// TwinCAT 3 PLC project las_bts
// Title: lcls-plc-las-bts
// Company: SLAC
// ProjectVersion: 1.0.0
// ProgramVersion: 3.1.4023.0
// libraries:
//   LCLSVacuumSerialDriverLib, * (SLAC)
//   Tc2_SerialCom, * (Beckhoff Automation GmbH)
//   Tc2_Standard, * (Beckhoff Automation GmbH)
//   Tc2_System, * (Beckhoff Automation GmbH)
//   Tc2_Utilities, * (Beckhoff Automation GmbH)
//   Tc3_Module, * (Beckhoff Automation GmbH)
//   TcUnit, * (www.tcunit.org)
//   LCLS General,2.4.2,SLAC
//   LCLS Vacuum,2.0.1,SLAC - LCLS
//   PMPS,2.2.1,SLAC - LCLS
// project tree:
//   / ComTask.TcTTO (not stored), PlcTask.TcTTO (not stored)
//   DUTs/ ST_ShutterControl.TcDUT (not stored), ST_SourceDataStore.TcDUT (not stored), ST_EpicsMotorMSTA.TcDUT (not stored)
//   GVLs/ GVL_BTPS.TcGVL (not stored), GVL_BTPS_Constants.TcGVL (not stored), GVL_BTPS_Retain.TcGVL (not stored), GVL_BTS_VAC.TcGVL, GVL_COM.TcGVL (not stored), GVL_Constants.TcGVL (not stored), GVL_Shutters.TcGVL (not stored), GVL_Variables.TcGVL (not stored)
//   POUs/BTPS/ FB_DestinationDataStore.TcPOU (not stored), FB_EpicsMotorMonitor.TcPOU (not stored), FB_EpicsStatsMonitor.TcPOU (not stored), FB_RangeComparison.TcPOU (not stored), FB_ShutterSafety.TcPOU (not stored), F_IsValveReady.TcPOU (not stored)
//   POUs/BTPS/Tests/ FB_TestRangeComparison.TcPOU (not stored), FB_TestShutterSafety.TcPOU (not stored), FB_Test_EpicsCentroidMonitor.TcPOU (not stored), FB_Test_EpicsMotorMonitor.TcPOU (not stored), PRG_RunTests.TcPOU (not stored)
//   POUs/ DIAGNOSTICS.TcPOU (not stored), MAIN.TcPOU (not stored), PRG_BTPS.TcPOU (not stored), PRG_COM.TcPOU (not stored), PRG_GAUGES.TcPOU (not stored), PRG_PUMPS.TcPOU (not stored), PRG_SavePeristentVariables.TcPOU (not stored), PRG_ShutterRequest.TcPOU (not stored), PRG_VALVES.TcPOU
// real-time tasks:
//   TASK PlcTask: cycle T#10ms, priority 20, ADS port 350
//   TASK ComTask: cycle T#11ms, priority 1, ADS port 351
// I/O:
//   DEVICE EtherCAT1
// variable links:
//   las_bts/las_bts Instance <-> EtherCAT1/EK1100_01_00/EL1004_01_16
//     PlcTask Inputs/GVL_BTS_VAC.fb_LS3_PIP.i_xSP_DI <-> Channel 1/Input
//     PlcTask Inputs/GVL_BTS_VAC.fb_LS4_PIP.i_xSP_DI <-> Channel 2/Input
//     PlcTask Inputs/GVL_BTS_VAC.fb_LS6_PIP.i_xSP_DI <-> Channel 3/Input
//   las_bts/las_bts Instance <-> EtherCAT1/EK1100_01_00/EL1124_01_06
//     PlcTask Inputs/GVL_BTS_VAC.fb_LS3_GCC.i_xDisc_Active <-> Channel 4/Input
//     PlcTask Inputs/GVL_BTS_VAC.fb_LS3_GCC.i_xHV_ON <-> Channel 3/Input
//     PlcTask Inputs/GVL_BTS_VAC.fb_PP_GCC.i_xDisc_Active <-> Channel 2/Input
//     PlcTask Inputs/GVL_BTS_VAC.fb_PP_GCC.i_xHV_ON <-> Channel 1/Input
//   las_bts/las_bts Instance <-> EtherCAT1/EK1100_01_00/EL1124_01_07
//     PlcTask Inputs/GVL_BTS_VAC.fb_DP_GCC.i_xDisc_Active <-> Channel 4/Input
//     PlcTask Inputs/GVL_BTS_VAC.fb_DP_GCC.i_xHV_ON <-> Channel 3/Input
//     PlcTask Inputs/GVL_BTS_VAC.fb_LD2_GCC.i_xDisc_Active <-> Channel 2/Input
//     PlcTask Inputs/GVL_BTS_VAC.fb_LD2_GCC.i_xHV_ON <-> Channel 1/Input
//   las_bts/las_bts Instance <-> EtherCAT1/EK1100_01_00/EL1124_01_08
//     PlcTask Inputs/GVL_BTS_VAC.fb_LD8_GCC.i_xDisc_Active <-> Channel 2/Input
//     PlcTask Inputs/GVL_BTS_VAC.fb_LD8_GCC.i_xHV_ON <-> Channel 1/Input
//     PlcTask Inputs/GVL_BTS_VAC.fb_LS4_GCC.i_xDisc_Active <-> Channel 4/Input
//     PlcTask Inputs/GVL_BTS_VAC.fb_LS4_GCC.i_xHV_ON <-> Channel 3/Input
//   las_bts/las_bts Instance <-> EtherCAT1/EK1100_01_00/EL2624_01_01
//     PlcTask Outputs/GVL_BTS_VAC.fb_LD8_GCC.q_xHV_DIS <-> Channel 1/Output
//     PlcTask Outputs/GVL_BTS_VAC.fb_LS3_GCC.q_xHV_DIS <-> Channel 3/Output
//     PlcTask Outputs/GVL_BTS_VAC.fb_LS4_GCC.q_xHV_DIS <-> Channel 4/Output
//   las_bts/las_bts Instance <-> EtherCAT1/EK1100_01_00/EL2624_01_02
//     PlcTask Outputs/GVL_BTS_VAC.fb_DP_GCC.q_xHV_DIS <-> Channel 4/Output
//     PlcTask Outputs/GVL_BTS_VAC.fb_LD2_GCC.q_xHV_DIS <-> Channel 1/Output
//     PlcTask Outputs/GVL_BTS_VAC.fb_PP_GCC.q_xHV_DIS <-> Channel 2/Output
//   las_bts/las_bts Instance <-> EtherCAT1/EK1100_01_00/EL2794_01_17
//     PlcTask Outputs/GVL_BTS_VAC.fb_LS3_PIP.q_xHVEna_DO <-> Channel 1/Output
//     PlcTask Outputs/GVL_BTS_VAC.fb_LS4_PIP.q_xHVEna_DO <-> Channel 2/Output
//     PlcTask Outputs/GVL_BTS_VAC.fb_LS6_PIP.q_xHVEna_DO <-> Channel 3/Output
//   las_bts/las_bts Instance <-> EtherCAT1/EK1100_01_00/EL3064_01_15
//     PlcTask Inputs/GVL_BTS_VAC.fb_LS3_PIP.i_iPRESS <-> AI Standard Channel 1/Value
//     PlcTask Inputs/GVL_BTS_VAC.fb_LS4_PIP.i_iPRESS <-> AI Standard Channel 2/Value
//     PlcTask Inputs/GVL_BTS_VAC.fb_LS6_PIP.i_iPRESS <-> AI Standard Channel 3/Value
//   las_bts/las_bts Instance <-> EtherCAT1/EK1100_01_00/EL3174_01_09
//     PlcTask Inputs/GVL_BTS_VAC.fb_DP_GCC.i_iPRESS_R <-> AI Standard Channel 4/Value
//     PlcTask Inputs/GVL_BTS_VAC.fb_LD2_GCC.i_iPRESS_R <-> AI Standard Channel 1/Value
//     PlcTask Inputs/GVL_BTS_VAC.fb_LS4_GPI.i_iPRESS_R <-> AI Standard Channel 3/Value
//     PlcTask Inputs/GVL_BTS_VAC.fb_LS6_GPI.i_iPRESS_R <-> AI Standard Channel 3/Value
//     PlcTask Inputs/GVL_BTS_VAC.fb_PP_GCC.i_iPRESS_R <-> AI Standard Channel 2/Value
//   las_bts/las_bts Instance <-> EtherCAT1/EK1100_01_00/EL3174_01_10
//     PlcTask Inputs/GVL_BTS_VAC.fb_DP_GPI.i_iPRESS_R <-> AI Standard Channel 2/Value
//     PlcTask Inputs/GVL_BTS_VAC.fb_LD2_GPI.i_iPRESS_R <-> AI Standard Channel 1/Value
//     PlcTask Inputs/GVL_BTS_VAC.fb_LS1_GPI.i_iPRESS_R <-> AI Standard Channel 4/Value
//     PlcTask Inputs/GVL_BTS_VAC.fb_PP_GPI_1.i_iPRESS_R <-> AI Standard Channel 3/Value
//   las_bts/las_bts Instance <-> EtherCAT1/EK1100_01_00/EL3174_01_11
//     PlcTask Inputs/GVL_BTS_VAC.fb_LD8_GCC.i_iPRESS_R <-> AI Standard Channel 3/Value
//     PlcTask Inputs/GVL_BTS_VAC.fb_LD8_GPI.i_iPRESS_R <-> AI Standard Channel 2/Value
//     PlcTask Inputs/GVL_BTS_VAC.fb_LS3_GPI.i_iPRESS_R <-> AI Standard Channel 4/Value
//     PlcTask Inputs/GVL_BTS_VAC.fb_PP_GPI_2.i_iPRESS_R <-> AI Standard Channel 1/Value
//   las_bts/las_bts Instance <-> EtherCAT1/EK1100_01_00/EL3174_01_8A
//     PlcTask Inputs/GVL_BTS_VAC.fb_LS3_GCC.i_iPRESS_R <-> AI Standard Channel 2/Value
//     PlcTask Inputs/GVL_BTS_VAC.fb_LS4_GCC.i_iPRESS_R <-> AI Standard Channel 3/Value
//   las_bts/las_bts Instance <-> EtherCAT1/EK1100_02_00/EL1002_02_01
//     PlcTask Inputs/GVL_BTS_VAC.fb_PP_VRC_1.i_xClsLS <-> Channel 1/Input
//     PlcTask Inputs/GVL_BTS_VAC.fb_PP_VRC_1.i_xOpnLS <-> Channel 2/Input
//   las_bts/las_bts Instance <-> EtherCAT1/EK1100_02_00/EL1002_02_03
//     PlcTask Inputs/GVL_BTS_VAC.fb_PP_VRC_3.i_xClsLS <-> Channel 1/Input
//     PlcTask Inputs/GVL_BTS_VAC.fb_PP_VRC_3.i_xOpnLS <-> Channel 2/Input
//   las_bts/las_bts Instance <-> EtherCAT1/EK1100_02_00/EL1004_02_06
//     PlcTask Inputs/GVL_BTS_VAC.fb_LD9_VGC.i_xClsLS <-> Channel 3/Input
//     PlcTask Inputs/GVL_BTS_VAC.fb_LD9_VGC.i_xOpnLS <-> Channel 4/Input
//     PlcTask Inputs/GVL_BTS_VAC.fb_LS1_VGC.i_xClsLS <-> Channel 1/Input
//     PlcTask Inputs/GVL_BTS_VAC.fb_LS1_VGC.i_xOpnLS <-> Channel 2/Input
//   las_bts/las_bts Instance <-> EtherCAT1/EK1100_02_00/EL1004_02_07
//     PlcTask Inputs/GVL_BTS_VAC.fb_LD10_VGC.i_xClsLS <-> Channel 1/Input
//     PlcTask Inputs/GVL_BTS_VAC.fb_LD8_VGC.i_xClsLS <-> Channel 3/Input
//     PlcTask Inputs/GVL_BTS_VAC.fb_LD10_VGC.i_xOpnLS <-> Channel 2/Input
//     PlcTask Inputs/GVL_BTS_VAC.fb_LD8_VGC.i_xOpnLS <-> Channel 4/Input
//   las_bts/las_bts Instance <-> EtherCAT1/EK1100_02_00/EL1004_02_09
//     PlcTask Inputs/GVL_BTS_VAC.fb_LS5_VGC.i_xClsLS <-> Channel 3/Input
//     PlcTask Inputs/GVL_BTS_VAC.fb_LS8_VGC.i_xClsLS <-> Channel 1/Input
//     PlcTask Inputs/GVL_BTS_VAC.fb_LS5_VGC.i_xOpnLS <-> Channel 4/Input
//     PlcTask Inputs/GVL_BTS_VAC.fb_LS8_VGC.i_xOpnLS <-> Channel 2/Input
//   las_bts/las_bts Instance <-> EtherCAT1/EK1100_02_00/EL1004_02_10
//     PlcTask Inputs/GVL_BTS_VAC.fb_LD14_VGC.i_xClsLS <-> Channel 3/Input
//     PlcTask Inputs/GVL_BTS_VAC.fb_LD4_VGC.i_xClsLS <-> Channel 1/Input
//     PlcTask Inputs/GVL_BTS_VAC.fb_LD14_VGC.i_xOpnLS <-> Channel 4/Input
//     PlcTask Inputs/GVL_BTS_VAC.fb_LD4_VGC.i_xOpnLS <-> Channel 2/Input
//   las_bts/las_bts Instance <-> EtherCAT1/EK1100_02_00/EL1004_02_12
//     PlcTask Inputs/GVL_BTS_VAC.fb_LD2_VGC.i_xClsLS <-> Channel 3/Input
//     PlcTask Inputs/GVL_BTS_VAC.fb_LD2_VGC.i_xOpnLS <-> Channel 4/Input
//     PlcTask Inputs/GVL_BTS_VAC.fb_PP_VGC.i_xClsLS <-> Channel 1/Input
//     PlcTask Inputs/GVL_BTS_VAC.fb_PP_VGC.i_xOpnLS <-> Channel 2/Input
//   las_bts/las_bts Instance <-> EtherCAT1/EK1100_02_00/EL1004_02_13
//     PlcTask Inputs/GVL_BTS_VAC.fb_LD6_VGC.i_xClsLS <-> Channel 3/Input
//     PlcTask Inputs/GVL_BTS_VAC.fb_LD6_VGC.i_xOpnLS <-> Channel 4/Input
//     PlcTask Inputs/GVL_BTS_VAC.fb_LS6_VGC.i_xClsLS <-> Channel 2/Input
//     PlcTask Inputs/GVL_BTS_VAC.fb_LS6_VGC.i_xOpnLS <-> Channel 1/Input
//   las_bts/las_bts Instance <-> EtherCAT1/EK1100_02_00/EL2004_02_04
//     PlcTask Outputs/GVL_BTS_VAC.fb_PP_VRC_1.q_xOPN_DO <-> Channel 1/Output
//     PlcTask Outputs/GVL_BTS_VAC.fb_PP_VRC_2.q_xOPN_DO <-> Channel 3/Output
//     PlcTask Outputs/GVL_BTS_VAC.fb_PP_VRC_3.q_xOPN_DO <-> Channel 4/Output
//   las_bts/las_bts Instance <-> EtherCAT1/EK1100_02_00/EL2004_02_05
//     PlcTask Outputs/GVL_BTS_VAC.fb_PP_VVC.q_xOPN_DO <-> Channel 3/Output
//     PlcTask Outputs/GVL_BTS_VAC.fb_VP_VVC_1.q_xOPN_DO <-> Channel 1/Output
//     PlcTask Outputs/GVL_BTS_VAC.fb_VP_VVC_2.q_xOPN_DO <-> Channel 2/Output
//   las_bts/las_bts Instance <-> EtherCAT1/EK1100_02_00/EL2004_02_08
//     PlcTask Outputs/GVL_BTS_VAC.fb_LD10_VGC.q_xOPN_DO <-> Channel 3/Output
//     PlcTask Outputs/GVL_BTS_VAC.fb_LD8_VGC.q_xOPN_DO <-> Channel 4/Output
//     PlcTask Outputs/GVL_BTS_VAC.fb_LD9_VGC.q_xOPN_DO <-> Channel 2/Output
//     PlcTask Outputs/GVL_BTS_VAC.fb_LS1_VGC.q_xOPN_DO <-> Channel 1/Output
//   las_bts/las_bts Instance <-> EtherCAT1/EK1100_02_00/EL2004_02_11
//     PlcTask Outputs/GVL_BTS_VAC.fb_LD14_VGC.q_xOPN_DO <-> Channel 4/Output
//     PlcTask Outputs/GVL_BTS_VAC.fb_LD4_VGC.q_xOPN_DO <-> Channel 1/Output
//     PlcTask Outputs/GVL_BTS_VAC.fb_LS5_VGC.q_xOPN_DO <-> Channel 2/Output
//     PlcTask Outputs/GVL_BTS_VAC.fb_LS8_VGC.q_xOPN_DO <-> Channel 3/Output
//   las_bts/las_bts Instance <-> EtherCAT1/EK1100_02_00/EL2004_02_14
//     PlcTask Outputs/GVL_BTS_VAC.fb_LD2_VGC.q_xOPN_DO <-> Channel 3/Output
//     PlcTask Outputs/GVL_BTS_VAC.fb_LD6_VGC.q_xOPN_DO <-> Channel 4/Output
//     PlcTask Outputs/GVL_BTS_VAC.fb_LS6_VGC.q_xOPN_DO <-> Channel 1/Output
//     PlcTask Outputs/GVL_BTS_VAC.fb_PP_VGC.q_xOPN_DO <-> Channel 2/Output
//   las_bts/las_bts Instance <-> EtherCAT1/EK1100_02_00/EL2004_02_15
//     PlcTask Outputs/GVL_BTS_VAC.fb_PP_VRC_4.q_xOPN_DO <-> Channel 2/Output
//     PlcTask Outputs/GVL_BTS_VAC.fb_VP_VVC_4.q_xOPN_DO <-> Channel 1/Output
//   las_bts/las_bts Instance <-> EtherCAT1/EK1100_02_00/EL3064_02_16
//     PlcTask Inputs/GVL_BTS_VAC.fb_LD6_GCC.i_iPRESS_R <-> AI Standard Channel 2/Value
//     PlcTask Inputs/GVL_BTS_VAC.fb_LS6_GCC.i_iPRESS_R <-> AI Standard Channel 1/Value
//   las_bts/las_bts Instance <-> EtherCAT1/EK1100_03_00/EL1004_03_17
//     PlcTask Inputs/GVL_BTS_VAC.fb_PP_VRC_4.i_xClsLS <-> Channel 2/Input
//     PlcTask Inputs/GVL_BTS_VAC.fb_PP_VRC_4.i_xOpnLS <-> Channel 1/Input
//   las_bts/las_bts Instance <-> EtherCAT1/EK1100_03_00/EL1124_03_06
//     PlcTask Inputs/GVL_BTS_VAC.fb_LD9_GCC.i_xDisc_Active <-> Channel 2/Input
//     PlcTask Inputs/GVL_BTS_VAC.fb_LD9_GCC.i_xHV_ON <-> Channel 1/Input
//     PlcTask Inputs/GVL_BTS_VAC.fb_LS1_GCC.i_xDisc_Active <-> Channel 4/Input
//     PlcTask Inputs/GVL_BTS_VAC.fb_LS1_GCC.i_xHV_ON <-> Channel 3/Input
//   las_bts/las_bts Instance <-> EtherCAT1/EK1100_03_00/EL1124_03_07
//     PlcTask Inputs/GVL_BTS_VAC.fb_LD10_GCC.i_xDisc_Active <-> Channel 4/Input
//     PlcTask Inputs/GVL_BTS_VAC.fb_LD14_GCC.i_xDisc_Active <-> Channel 2/Input
//     PlcTask Inputs/GVL_BTS_VAC.fb_LD10_GCC.i_xHV_ON <-> Channel 3/Input
//     PlcTask Inputs/GVL_BTS_VAC.fb_LD14_GCC.i_xHV_ON <-> Channel 1/Input
//   las_bts/las_bts Instance <-> EtherCAT1/EK1100_03_00/EL1124_03_08
//     PlcTask Inputs/GVL_BTS_VAC.fb_LS5_GCC.i_xDisc_Active <-> Channel 2/Input
//     PlcTask Inputs/GVL_BTS_VAC.fb_LS8_GCC.i_xDisc_Active <-> Channel 4/Input
//     PlcTask Inputs/GVL_BTS_VAC.fb_LS5_GCC.i_xHV_ON <-> Channel 1/Input
//     PlcTask Inputs/GVL_BTS_VAC.fb_LS8_GCC.i_xHV_ON <-> Channel 3/Input
//   las_bts/las_bts Instance <-> EtherCAT1/EK1100_03_00/EL1124_03_09
//     PlcTask Inputs/GVL_BTS_VAC.fb_LD4_GCC.i_xDisc_Active <-> Channel 4/Input
//     PlcTask Inputs/GVL_BTS_VAC.fb_LD4_GCC.i_xHV_ON <-> Channel 3/Input
//   las_bts/las_bts Instance <-> EtherCAT1/EK1100_03_00/EL2624_03_01
//     PlcTask Outputs/GVL_BTS_VAC.fb_LD10_GCC.q_xHV_DIS <-> Channel 2/Output
//     PlcTask Outputs/GVL_BTS_VAC.fb_LD14_GCC.q_xHV_DIS <-> Channel 3/Output
//     PlcTask Outputs/GVL_BTS_VAC.fb_LD9_GCC.q_xHV_DIS <-> Channel 1/Output
//     PlcTask Outputs/GVL_BTS_VAC.fb_LS1_GCC.q_xHV_DIS <-> Channel 4/Output
//   las_bts/las_bts Instance <-> EtherCAT1/EK1100_03_00/EL2624_03_02
//     PlcTask Outputs/GVL_BTS_VAC.fb_LD4_GCC.q_xHV_DIS <-> Channel 4/Output
//     PlcTask Outputs/GVL_BTS_VAC.fb_LS5_GCC.q_xHV_DIS <-> Channel 1/Output
//     PlcTask Outputs/GVL_BTS_VAC.fb_LS8_GCC.q_xHV_DIS <-> Channel 2/Output
//   las_bts/las_bts Instance <-> EtherCAT1/EK1100_03_00/EL3174_03_10
//     PlcTask Inputs/GVL_BTS_VAC.fb_LD10_GCC.i_iPRESS_R <-> AI Standard Channel 2/Value
//     PlcTask Inputs/GVL_BTS_VAC.fb_LD14_GCC.i_iPRESS_R <-> AI Standard Channel 3/Value
//     PlcTask Inputs/GVL_BTS_VAC.fb_LD9_GCC.i_iPRESS_R <-> AI Standard Channel 1/Value
//     PlcTask Inputs/GVL_BTS_VAC.fb_LS1_GCC.i_iPRESS_R <-> AI Standard Channel 4/Value
//   las_bts/las_bts Instance <-> EtherCAT1/EK1100_03_00/EL3174_03_11
//     PlcTask Inputs/GVL_BTS_VAC.fb_LD4_GCC.i_iPRESS_R <-> AI Standard Channel 4/Value
//     PlcTask Inputs/GVL_BTS_VAC.fb_LS5_GCC.i_iPRESS_R <-> AI Standard Channel 1/Value
//     PlcTask Inputs/GVL_BTS_VAC.fb_LS8_GCC.i_iPRESS_R <-> AI Standard Channel 2/Value
//   las_bts/las_bts Instance <-> EtherCAT1/EK1100_03_00/EL3174_03_12
//     PlcTask Inputs/GVL_BTS_VAC.fb_LD10_GPI.i_iPRESS_R <-> AI Standard Channel 2/Value
//     PlcTask Inputs/GVL_BTS_VAC.fb_LD14_GPI.i_iPRESS_R <-> AI Standard Channel 3/Value
//     PlcTask Inputs/GVL_BTS_VAC.fb_LD9_GPI.i_iPRESS_R <-> AI Standard Channel 1/Value
//   las_bts/las_bts Instance <-> EtherCAT1/EK1100_03_00/EL3174_03_13
//     PlcTask Inputs/GVL_BTS_VAC.fb_LD4_GPI.i_iPRESS_R <-> AI Standard Channel 4/Value
//     PlcTask Inputs/GVL_BTS_VAC.fb_LD6_GPI.i_iPRESS_R <-> AI Standard Channel 3/Value
//     PlcTask Inputs/GVL_BTS_VAC.fb_LS5_GPI.i_iPRESS_R <-> AI Standard Channel 1/Value
//     PlcTask Inputs/GVL_BTS_VAC.fb_LS8_GPI.i_iPRESS_R <-> AI Standard Channel 2/Value
//   las_bts/las_bts Instance <-> EtherCAT1/EK1100_04_00/EL1004_04_02
//     PlcTask Inputs/GVL_Shutters.fbLS1.bCloseStatus <-> Channel 2/Input
//     PlcTask Inputs/GVL_Shutters.fbLS4.bCloseStatus <-> Channel 4/Input
//     PlcTask Inputs/GVL_Shutters.fbLS1.bOpenStatus <-> Channel 1/Input
//     PlcTask Inputs/GVL_Shutters.fbLS4.bOpenStatus <-> Channel 3/Input
//   las_bts/las_bts Instance <-> EtherCAT1/EK1100_04_00/EL1004_04_03
//     PlcTask Inputs/GVL_Shutters.fbLS5.bCloseStatus <-> Channel 2/Input
//     PlcTask Inputs/GVL_Shutters.fbLS8.bCloseStatus <-> Channel 4/Input
//     PlcTask Inputs/GVL_Shutters.fbLS5.bOpenStatus <-> Channel 1/Input
//     PlcTask Inputs/GVL_Shutters.fbLS8.bOpenStatus <-> Channel 3/Input
//   las_bts/las_bts Instance <-> EtherCAT1/EK1100_04_00/EL1004_04_04
//     PlcTask Inputs/GVL_Shutters.fbLS1.bLssStatus <-> Channel 1/Input
//     PlcTask Inputs/GVL_Shutters.fbLS4.bLssStatus <-> Channel 2/Input
//     PlcTask Inputs/GVL_Shutters.fbLS5.bLssStatus <-> Channel 3/Input
//     PlcTask Inputs/GVL_Shutters.fbLS8.bLssStatus <-> Channel 4/Input
//   las_bts/las_bts Instance <-> EtherCAT1/EK1100_04_00/EL1004_04_06
//     PlcTask Inputs/GVL_Shutters.fbLS3.bCloseStatus <-> Channel 2/Input
//     PlcTask Inputs/GVL_Shutters.fbLS6.bCloseStatus <-> Channel 4/Input
//     PlcTask Inputs/GVL_Shutters.fbLS3.bOpenStatus <-> Channel 1/Input
//     PlcTask Inputs/GVL_Shutters.fbLS6.bOpenStatus <-> Channel 3/Input
//   las_bts/las_bts Instance <-> EtherCAT1/EK1100_04_00/EL1004_04_07
//     PlcTask Inputs/GVL_Shutters.fbLS3.bLssStatus <-> Channel 1/Input
//     PlcTask Inputs/GVL_Shutters.fbLS6.bLssStatus <-> Channel 2/Input
//   las_bts/las_bts Instance <-> EtherCAT1/EK1100_04_00/EL2624_04_01
//     PlcTask Outputs/GVL_Shutters.fbLS1.bOpenRequest <-> Channel 1/Output
//     PlcTask Outputs/GVL_Shutters.fbLS4.bOpenRequest <-> Channel 2/Output
//     PlcTask Outputs/GVL_Shutters.fbLS5.bOpenRequest <-> Channel 3/Output
//     PlcTask Outputs/GVL_Shutters.fbLS8.bOpenRequest <-> Channel 4/Output
//   las_bts/las_bts Instance <-> EtherCAT1/EK1100_04_00/EL2624_04_05
//     PlcTask Outputs/GVL_Shutters.fbLS3.bOpenRequest <-> Channel 1/Output
//     PlcTask Outputs/GVL_Shutters.fbLS6.bOpenRequest <-> Channel 3/Output
//   las_bts/las_bts Instance <-> EtherCAT1/EK1200_00_00/EL1004_00_01
//     PlcTask Inputs/GVL_BTS_VAC.fb_PP_PMF.i_xAlarm <-> Channel 3/Input
//     PlcTask Inputs/GVL_BTS_VAC.fb_PP_PMF.i_xIsRun <-> Channel 1/Input
//     PlcTask Inputs/GVL_BTS_VAC.fb_PP_PMF.i_xRemote <-> Channel 2/Input
//     PlcTask Inputs/GVL_BTS_VAC.fb_PP_PMF.i_xWarning <-> Channel 4/Input
//   las_bts/las_bts Instance <-> EtherCAT1/EK1200_00_00/EL1004_00_03
//     PlcTask Inputs/GVL_BTS_VAC.fb_PP_PTM.i_xAtSpd <-> Channel 3/Input
//     PlcTask Inputs/GVL_BTS_VAC.fb_PP_PTM.i_xFaultNC <-> Channel 1/Input
//     PlcTask Inputs/GVL_BTS_VAC.fb_PP_PTM.i_xRemote <-> Channel 2/Input
//   las_bts/las_bts Instance <-> EtherCAT1/EK1200_00_00/EL1004_00_07
//     PlcTask Inputs/GVL_BTS_VAC.fb_LD2_PIP.i_xSP_DI <-> Channel 1/Input
//     PlcTask Inputs/GVL_BTS_VAC.fb_LD8_PIP.i_xSP_DI <-> Channel 4/Input
//     PlcTask Inputs/GVL_BTS_VAC.fb_LS1_PIP.i_xSP_DI <-> Channel 2/Input
//     PlcTask Inputs/GVL_BTS_VAC.fb_PP_PIP.i_xSP_DI <-> Channel 3/Input
//   las_bts/las_bts Instance <-> EtherCAT1/EK1200_00_00/EL1004_00_10
//     PlcTask Inputs/GVL_BTS_VAC.fb_LD4_PIP.i_xSP_DI <-> Channel 1/Input
//     PlcTask Inputs/GVL_BTS_VAC.fb_LD6_PIP.i_xSP_DI <-> Channel 2/Input
//     PlcTask Inputs/GVL_BTS_VAC.fb_LS5_PIP.i_xSP_DI <-> Channel 4/Input
//     PlcTask Inputs/GVL_BTS_VAC.fb_LS8_PIP.i_xSP_DI <-> Channel 3/Input
//   las_bts/las_bts Instance <-> EtherCAT1/EK1200_00_00/EL1004_00_13
//     PlcTask Inputs/GVL_BTS_VAC.fb_LD10_PIP.i_xSP_DI <-> Channel 1/Input
//     PlcTask Inputs/GVL_BTS_VAC.fb_LD14_PIP.i_xSP_DI <-> Channel 3/Input
//     PlcTask Inputs/GVL_BTS_VAC.fb_LD9_PIP.i_xSP_DI <-> Channel 2/Input
//   las_bts/las_bts Instance <-> EtherCAT1/EK1200_00_00/EL1004_00_16
//     PlcTask Inputs/GVL_BTS_VAC.fb_LS3_VGC.i_xClsLS <-> Channel 2/Input
//     PlcTask Inputs/GVL_BTS_VAC.fb_LS4_VGC.i_xClsLS <-> Channel 4/Input
//     PlcTask Inputs/GVL_BTS_VAC.fb_LS3_VGC.i_xOpnLS <-> Channel 1/Input
//     PlcTask Inputs/GVL_BTS_VAC.fb_LS4_VGC.i_xOpnLS <-> Channel 3/Input
//   las_bts/las_bts Instance <-> EtherCAT1/EK1200_00_00/EL2004_00_04
//     PlcTask Outputs/GVL_BTS_VAC.fb_PP_PTM.q_PumpingStation <-> Channel 3/Output
//     PlcTask Outputs/GVL_BTS_VAC.fb_PP_PTM.q_RunDO <-> Channel 1/Output
//     PlcTask Outputs/GVL_BTS_VAC.fb_PP_PTM.q_xRemote <-> Channel 2/Output
//   las_bts/las_bts Instance <-> EtherCAT1/EK1200_00_00/EL2004_00_17
//     PlcTask Outputs/GVL_BTS_VAC.fb_LS3_VGC.q_xOPN_DO <-> Channel 1/Output
//     PlcTask Outputs/GVL_BTS_VAC.fb_LS4_VGC.q_xOPN_DO <-> Channel 2/Output
//   las_bts/las_bts Instance <-> EtherCAT1/EK1200_00_00/EL2794_00_02
//     PlcTask Outputs/GVL_BTS_VAC.fb_PP_PMF.q_xLspdDo <-> Channel 2/Output
//     PlcTask Outputs/GVL_BTS_VAC.fb_PP_PMF.q_xResetDo <-> Channel 3/Output
//     PlcTask Outputs/GVL_BTS_VAC.fb_PP_PMF.q_xRunDO <-> Channel 1/Output
//   las_bts/las_bts Instance <-> EtherCAT1/EK1200_00_00/EL2794_00_06
//     PlcTask Outputs/GVL_BTS_VAC.fb_LD2_PIP.q_xHVEna_DO <-> Channel 1/Output
//     PlcTask Outputs/GVL_BTS_VAC.fb_LD8_PIP.q_xHVEna_DO <-> Channel 4/Output
//     PlcTask Outputs/GVL_BTS_VAC.fb_LS1_PIP.q_xHVEna_DO <-> Channel 2/Output
//     PlcTask Outputs/GVL_BTS_VAC.fb_PP_PIP.q_xHVEna_DO <-> Channel 3/Output
//   las_bts/las_bts Instance <-> EtherCAT1/EK1200_00_00/EL2794_00_09
//     PlcTask Outputs/GVL_BTS_VAC.fb_LD4_PIP.q_xHVEna_DO <-> Channel 1/Output
//     PlcTask Outputs/GVL_BTS_VAC.fb_LD6_PIP.q_xHVEna_DO <-> Channel 2/Output
//     PlcTask Outputs/GVL_BTS_VAC.fb_LS5_PIP.q_xHVEna_DO <-> Channel 4/Output
//     PlcTask Outputs/GVL_BTS_VAC.fb_LS8_PIP.q_xHVEna_DO <-> Channel 3/Output
//   las_bts/las_bts Instance <-> EtherCAT1/EK1200_00_00/EL2794_00_12
//     PlcTask Outputs/GVL_BTS_VAC.fb_LD10_PIP.q_xHVEna_DO <-> Channel 1/Output
//     PlcTask Outputs/GVL_BTS_VAC.fb_LD14_PIP.q_xHVEna_DO <-> Channel 3/Output
//     PlcTask Outputs/GVL_BTS_VAC.fb_LD9_PIP.q_xHVEna_DO <-> Channel 2/Output
//   las_bts/las_bts Instance <-> EtherCAT1/EK1200_00_00/EL3064_00_08
//     PlcTask Inputs/GVL_BTS_VAC.fb_LD2_PIP.i_iPRESS <-> AI Standard Channel 1/Value
//     PlcTask Inputs/GVL_BTS_VAC.fb_LD8_PIP.i_iPRESS <-> AI Standard Channel 4/Value
//     PlcTask Inputs/GVL_BTS_VAC.fb_LS1_PIP.i_iPRESS <-> AI Standard Channel 2/Value
//     PlcTask Inputs/GVL_BTS_VAC.fb_PP_PIP.i_iPRESS <-> AI Standard Channel 3/Value
//   las_bts/las_bts Instance <-> EtherCAT1/EK1200_00_00/EL3064_00_11
//     PlcTask Inputs/GVL_BTS_VAC.fb_LD4_PIP.i_iPRESS <-> AI Standard Channel 1/Value
//     PlcTask Inputs/GVL_BTS_VAC.fb_LD6_PIP.i_iPRESS <-> AI Standard Channel 2/Value
//     PlcTask Inputs/GVL_BTS_VAC.fb_LS5_PIP.i_iPRESS <-> AI Standard Channel 4/Value
//     PlcTask Inputs/GVL_BTS_VAC.fb_LS8_PIP.i_iPRESS <-> AI Standard Channel 3/Value
//   las_bts/las_bts Instance <-> EtherCAT1/EK1200_00_00/EL3064_00_14
//     PlcTask Inputs/GVL_BTS_VAC.fb_LD10_PIP.i_iPRESS <-> AI Standard Channel 1/Value
//     PlcTask Inputs/GVL_BTS_VAC.fb_LD14_PIP.i_iPRESS <-> AI Standard Channel 3/Value
//     PlcTask Inputs/GVL_BTS_VAC.fb_LD9_PIP.i_iPRESS <-> AI Standard Channel 2/Value
//   las_bts/las_bts Instance <-> EtherCAT1/EK1200_00_00/EL6021_00_05
//     ComTask Inputs/GVL_COM.PTM_stComIn/D[{0..21}] <-> COM TxPDO-Map Inputs/Data In {0..21}  (22 links)
//     ComTask Outputs/GVL_COM.PTM_stComOut/Ctrl <-> COM RxPDO-Map Outputs/Ctrl
//     ComTask Outputs/GVL_COM.PTM_stComOut/D[{0..21}] <-> COM RxPDO-Map Outputs/Data Out {0..21}  (22 links)

// ---- GVLs/GVL_BTS_VAC.TcGVL
//{attribute 'qualified_only'}
VAR_GLOBAL
    (* Valves *)
    g_FFOut : FB_HardwareFFOutput;

    {attribute 'pytmc'	  :=	' pv: LXLHN:VGC:01 '}
    {attribute 'TcLinkTo' := 	'.i_xOpnLS			:=	TIIB[EL1004_02_12]^Channel 2^Input;
                                 .i_xClsLS			:=	TIIB[EL1004_02_12]^Channel 1^Input;
                                 .q_xOPN_DO			:=	TIIB[EL2004_02_14]^Channel 2^Output'}
    fb_PP_VGC : FB_VGC; // Gate valve, vacuum switchbox

    {attribute 'pytmc' 	  :=	' pv: LXLHN:VVC:01 '}
    {attribute 'TcLinkTo' := 	'.q_xOPN_DO			:=	TIIB[EL2004_02_05]^Channel 3^Output'}
    fb_PP_VVC : FB_VVC; // Turbo N2 purge


    {attribute 'pytmc'	  :=	' pv: LXLHN:VRC:01 '}
    {attribute 'TcLinkTo' := 	'.i_xOpnLS			:=	TIIB[EL1002_02_01]^Channel 2^Input;
                                 .i_xClsLS			:=	TIIB[EL1002_02_01]^Channel 1^Input;
                                 .q_xOPN_DO			:=	TIIB[EL2004_02_04]^Channel 1^Output'}
    fb_PP_VRC_1 : FB_VRC; // O-ring diff pump valve

    {attribute 'pytmc'	  :=	' pv: LXLHN:VRC:02 '}
    {attribute 'TcLinkTo' := 	'.q_xOPN_DO			:=	TIIB[EL2004_02_04]^Channel 3^Output'}
                                (*'.i_xOpnLS			:=	TIIB[EL1002_02_02]^Channel 2^Input;
                                 .i_xClsLS			:=	TIIB[EL1002_02_02]^Channel 1^Input;
                                 .q_xOPN_DO			:=	TIIB[EL2004_02_04]^Channel 3^Output'}		*)
    fb_PP_VRC_2 : FB_VVC; // Foreline valve //valve has bad readouts so using VVC

    {attribute 'pytmc'	  :=	' pv: LXLHN:VRC:03 '}
    {attribute 'TcLinkTo' := 	'.i_xOpnLS			:=	TIIB[EL1002_02_03]^Channel 2^Input;
                                 .i_xClsLS			:=	TIIB[EL1002_02_03]^Channel 1^Input;
                                 .q_xOPN_DO			:=	TIIB[EL2004_02_04]^Channel 4^Output'}
    fb_PP_VRC_3 : FB_VRC; // Slow pump valve

    st_VP_VVC_1 : ST_VVC;
    {attribute 'pytmc' 	  :=	' pv: LXLHN:VVC:02 '}
    {attribute 'TcLinkTo' := 	'.q_xOPN_DO			:=	TIIB[EL2004_02_05]^Channel 1^Output'}
    fb_VP_VVC_1 : FB_VVC; // Vent valve, Switchbox

    st_VP_VVC_2 : ST_VVC;
    {attribute 'pytmc' 	  :=	' pv: LXLHN:VVC:03 '}
    {attribute 'TcLinkTo' := 	'.q_xOPN_DO			:=	TIIB[EL2004_02_05]^Channel 2^Output'}
    fb_VP_VVC_2 : FB_VVC; // Vent valve, Slow, Switchbox

// Vent Valve addition
    st_VP_VVC_4 : ST_VVC;
    {attribute 'pytmc' 	  :=	' pv: LXLHN:VVC:04 '}
    {attribute 'TcLinkTo' := 	'.q_xOPN_DO			:=	TIIB[EL2004_02_15]^Channel 1^Output'}
    fb_VP_VVC_4 : FB_VVC;

    {attribute 'pytmc' 	  :=	' pv: LXLHN:VRC:04 '}
    {attribute 'TcLinkTo' := 	'.q_xOPN_DO			:=	TIIB[EL2004_02_15]^Channel 2^Output;
                                 .i_xOpnLS			:=	TIIB[EL1004_03_17]^Channel 1^Input;
                                 .i_xClsLS			:=	TIIB[EL1004_03_17]^Channel 2^Input'}
    fb_PP_VRC_4 : FB_VRC; // Turbo Isolation Valve


    (* Pumps *)
    {attribute 'pytmc' 	  := '
        pv: LXLHN:PTM:01
        io: io
    '}
    {attribute 'TcLinkTo' := 	'.i_xAtSpd			:=	TIIB[EL1004_00_03]^Channel 3^Input;
                                 .i_xRemote			:=	TIIB[EL1004_00_03]^Channel 2^Input;
                                 .i_xFaultNC		:=	TIIB[EL1004_00_03]^Channel 1^Input;
                                 .q_RunDO			:=	TIIB[EL2004_00_04]^Channel 1^Output;
                                 .q_xRemote			:=	TIIB[EL2004_00_04]^Channel 2^Output;
                                 .q_PumpingStation	:=	TIIB[EL2004_00_04]^Channel 3^Output'}
    fb_PP_PTM : FB_PTM_Pfeiffer; // Turbo pump

    // Serial port
    st_Pfeiffer_CTRL_PTM		: ARRAY[1..20] OF ST_PfeifferControl;
    st_Pfeiffer_RBK_PTM			: ARRAY[1..20] OF ST_PfeifferStatus;
    PTM_COM 					: FB_PFEIFFER_COM;

    {attribute 'pytmc' 	  := '
        pv: LXLHN:PMF:01
        io: io
    '}
    {attribute 'TcLinkTo' := 	'.i_xWarning		:=	TIIB[EL1004_00_01]^Channel 4^Input;
                                 .i_xAlarm			:=	TIIB[EL1004_00_01]^Channel 3^Input;
                                 .i_xRemote			:=	TIIB[EL1004_00_01]^Channel 2^Input;
                                 .i_xIsRun			:=	TIIB[EL1004_00_01]^Channel 1^Input;
                                 .q_xRunDO			:=	TIIB[EL2794_00_02]^Channel 1^Output;
                                 .q_xLspdDO			:=	TIIB[EL2794_00_02]^Channel 2^Output;
                                 .q_xResetDo		:=	TIIB[EL2794_00_02]^Channel 3^Output'}
    fb_PP_PMF : FB_KashiyamaPump; // Roughing Pump

    {attribute 'pytmc'    := 	' pv: LXLHN:PIP:01'}
    {attribute 'TcLinkTo' := 	'.i_iPRESS			:=	TIIB[EL3064_00_08]^AI Standard Channel 3^Value;
                                 .i_xSP_DI			:= 	TIIB[EL1004_00_07]^Channel 3^Input;
                                 .q_xHVEna_DO		:= 	TIIB[EL2794_00_06]^Channel 3^Output'}
    fb_PP_PIP : FB_PIP_Gamma; // Ion Pump, SW

    (* Gauges *)
    {attribute 'pytmc' 	  :=	' pv: LXLHN:GPI:01 '}
    {attribute 'TcLinkTo' := 	'.i_iPRESS_R		:=	TIIB[EL3174_01_10]^AI Standard Channel 3^Value '}
    fb_PP_GPI_1 : FB_MKS275; // Switchbox pumpline ATM gauge

    {attribute 'pytmc' 	  :=	' pv: LXLHN:GPI:02 '}
    {attribute 'TcLinkTo' := 	'.i_iPRESS_R		:=	TIIB[EL3174_01_11]^AI Standard Channel 1^Value '}
    fb_PP_GPI_2 : FB_MKS275; // Foreline gauge

    {attribute 'pytmc' 	  :=	' pv: LXLHN:GPI:03 '}
    {attribute 'TcLinkTo' := 	'.i_iPRESS_R		:=	TIIB[EL3174_01_10]^AI Standard Channel 2^Value '}
    fb_DP_GPI : FB_MKS275; // Switchbox gauge

    {attribute 'pytmc' 	  :=	' pv: LXLHN:GCC:01 '}
    {attribute 'TcLinkTo' := 	'.i_iPRESS_R		:=	TIIB[EL3174_01_09]^AI Standard Channel 2^Value;
                                 .i_xHV_ON	    	:=	TIIB[EL1124_01_06]^Channel 1^Input;
                                 .i_xDisc_Active	:=	TIIB[EL1124_01_06]^Channel 2^Input;
                                 .q_xHV_DIS			:= 	TIIB[EL2624_01_02]^Channel 2^Output	'}
    fb_PP_GCC : FB_MKS500; // Switchbox pumpline Cold Cathode gauge

    {attribute 'pytmc' 	  :=	' pv: LXLHN:GCC:02 '}
    {attribute 'TcLinkTo' := 	'.i_iPRESS_R		:=	TIIB[EL3174_01_09]^AI Standard Channel 4^Value;
                                 .i_xHV_ON	    	:=	TIIB[EL1124_01_07]^Channel 3^Input;
                                 .i_xDisc_Active	:=	TIIB[EL1124_01_07]^Channel 4^Input;
                                 .q_xHV_DIS			:= 	TIIB[EL2624_01_02]^Channel 4^Output	'}
    fb_DP_GCC : FB_MKS500; // Switchbox Cold Cathode gauge

    (* Transport Tubes *)
    // LS1
    {attribute 'pytmc'	  :=	' pv: LTLHN:LS1:VGC:01 '}
    {attribute 'TcLinkTo' := 	'.i_xOpnLS			:=	TIIB[EL1004_02_06]^Channel 2^Input;
                                 .i_xClsLS			:=	TIIB[EL1004_02_06]^Channel 1^Input;
                                 .q_xOPN_DO			:=	TIIB[EL2004_02_08]^Channel 1^Output'}
    fb_LS1_VGC : FB_VGC; // Gate valve, Input LS1 laser Table
    {attribute 'pytmc'    := 	' pv: LTLHN:LS1:PIP:01 '}
    {attribute 'TcLinkTo' := 	'.i_iPRESS			:=	TIIB[EL3064_00_08]^AI Standard Channel 2^Value;
                                 .i_xSP_DI			:= 	TIIB[EL1004_00_07]^Channel 2^Input;
                                 .q_xHVEna_DO		:= 	TIIB[EL2794_00_06]^Channel 2^Output'}
    fb_LS1_PIP : FB_PIP_Gamma; // Ion Pump, input tube LS1
    {attribute 'pytmc' 	  :=	' pv: LTLHN:LS1:GPI:01 '}
    {attribute 'TcLinkTo' := 	'.i_iPRESS_R		:=	TIIB[EL3174_01_10]^AI Standard Channel 4^Value '}
    fb_LS1_GPI : FB_MKS275; // Input tube LS1 ATM gauge
    {attribute 'pytmc' 	  :=	' pv: LTLHN:LS1:GCC:01 '}
    {attribute 'TcLinkTo' := 	'.i_iPRESS_R		:=	TIIB[EL3174_03_10]^AI Standard Channel 4^Value;
                                 .i_xHV_ON	    	:=	TIIB[EL1124_03_06]^Channel 3^Input;
                                 .i_xDisc_Active	:=	TIIB[EL1124_03_06]^Channel 4^Input;
                                 .q_xHV_DIS			:= 	TIIB[EL2624_03_01]^Channel 4^Output	'}
    fb_LS1_GCC : FB_MKS500; // Input tube LS1, Cold Cathode gauge

    // LS5
    {attribute 'pytmc'	  :=	' pv: LTLHN:LS5:VGC:01 '}
    {attribute 'TcLinkTo' := 	'.i_xOpnLS			:=	TIIB[EL1004_02_09]^Channel 4^Input;
                                 .i_xClsLS			:=	TIIB[EL1004_02_09]^Channel 3^Input;
                                 .q_xOPN_DO			:=	TIIB[EL2004_02_11]^Channel 2^Output'}
    fb_LS5_VGC : FB_VGC; // Gate valve, Input LS5 laser Table
    {attribute 'pytmc'    := 	' pv: LTLHN:LS5:PIP:01 '}
    {attribute 'TcLinkTo' := 	'.i_iPRESS			:=	TIIB[EL3064_00_11]^AI Standard Channel 4^Value;
                                 .i_xSP_DI			:= 	TIIB[EL1004_00_10]^Channel 4^Input;
                                 .q_xHVEna_DO		:= 	TIIB[EL2794_00_09]^Channel 4^Output'}
    fb_LS5_PIP : FB_PIP_Gamma; // Ion Pump, input tube LS5
    {attribute 'pytmc' 	  :=	' pv: LTLHN:LS5:GPI:01 '}
    {attribute 'TcLinkTo' := 	'.i_iPRESS_R		:=	TIIB[EL3174_03_13]^AI Standard Channel 1^Value '}
    fb_LS5_GPI : FB_MKS275; // Input tube LS5 ATM gauge
    {attribute 'pytmc' 	  :=	' pv: LTLHN:LS5:GCC:01 '}
    {attribute 'TcLinkTo' := 	'.i_iPRESS_R		:=	TIIB[EL3174_03_11]^AI Standard Channel 1^Value;
                                 .i_xHV_ON	    	:=	TIIB[EL1124_03_08]^Channel 1^Input;
                                 .i_xDisc_Active	:=	TIIB[EL1124_03_08]^Channel 2^Input;
                                 .q_xHV_DIS			:= 	TIIB[EL2624_03_02]^Channel 1^Output	'}
    fb_LS5_GCC : FB_MKS500; // Input tube LS5, Cold Cathode gauge

    // LS8
    {attribute 'pytmc'	  :=	' pv: LTLHN:LS8:VGC:01 '}
    {attribute 'TcLinkTo' := 	'.i_xOpnLS			:=	TIIB[EL1004_02_09]^Channel 2^Input;
                                 .i_xClsLS			:=	TIIB[EL1004_02_09]^Channel 1^Input;
                                 .q_xOPN_DO			:=	TIIB[EL2004_02_11]^Channel 3^Output'}
    fb_LS8_VGC : FB_VGC; // Gate valve, Input LS8 laser Table
    {attribute 'pytmc'    := 	' pv: LTLHN:LS8:PIP:01 '}
    {attribute 'TcLinkTo' := 	'.i_iPRESS			:=	TIIB[EL3064_00_11]^AI Standard Channel 3^Value;
                                 .i_xSP_DI			:= 	TIIB[EL1004_00_10]^Channel 3^Input;
                                 .q_xHVEna_DO		:= 	TIIB[EL2794_00_09]^Channel 3^Output'}
    fb_LS8_PIP : FB_PIP_Gamma; // Ion Pump, input tube LS8
    {attribute 'pytmc' 	  :=	' pv: LTLHN:LS8:GPI:01 '}
    {attribute 'TcLinkTo' := 	'.i_iPRESS_R		:=	TIIB[EL3174_03_13]^AI Standard Channel 2^Value '}
    fb_LS8_GPI : FB_MKS275; // Input tube LS8 ATM gauge
    {attribute 'pytmc' 	  :=	' pv: LTLHN:LS8:GCC:01 '}
    {attribute 'TcLinkTo' := 	'.i_iPRESS_R		:=	TIIB[EL3174_03_11]^AI Standard Channel 2^Value;
                                 .i_xHV_ON	    	:=	TIIB[EL1124_03_08]^Channel 3^Input;
                                 .i_xDisc_Active	:=	TIIB[EL1124_03_08]^Channel 4^Input;
                                 .q_xHV_DIS			:= 	TIIB[EL2624_03_02]^Channel 2^Output	'}
    fb_LS8_GCC : FB_MKS500; // Input tube LS8, Cold Cathode gauge

    // LD2
    {attribute 'pytmc'	  :=	' pv: LTLHN:LD2:VGC:01 '}
    {attribute 'TcLinkTo' := 	'.i_xOpnLS			:=	TIIB[EL1004_02_12]^Channel 4^Input;
                                 .i_xClsLS			:=	TIIB[EL1004_02_12]^Channel 3^Input;
                                 .q_xOPN_DO			:=	TIIB[EL2004_02_14]^Channel 3^Output'}
    fb_LD2_VGC : FB_VGC; // Gate valve, Output tube LD2 laser Table
    {attribute 'pytmc'    := 	' pv: LTLHN:LD2:PIP:01 '}
    {attribute 'TcLinkTo' := 	'.i_iPRESS			:=	TIIB[EL3064_00_08]^AI Standard Channel 1^Value;
                                 .i_xSP_DI			:= 	TIIB[EL1004_00_07]^Channel 1^Input;
                                 .q_xHVEna_DO		:= 	TIIB[EL2794_00_06]^Channel 1^Output'}
    fb_LD2_PIP : FB_PIP_Gamma; // Ion Pump, output tube LD2
    {attribute 'pytmc' 	  :=	' pv: LTLHN:LD2:GPI:01 '}
    {attribute 'TcLinkTo' := 	'.i_iPRESS_R		:=	TIIB[EL3174_01_10]^AI Standard Channel 1^Value '}
    fb_LD2_GPI : FB_MKS275; // Output tube LD2 ATM gauge
    {attribute 'pytmc' 	  :=	' pv: LTLHN:LD2:GCC:01 '}
    {attribute 'TcLinkTo' := 	'.i_iPRESS_R		:=	TIIB[EL3174_01_09]^AI Standard Channel 1^Value;
                                 .i_xHV_ON	    	:=	TIIB[EL1124_01_07]^Channel 1^Input;
                                 .i_xDisc_Active	:=	TIIB[EL1124_01_07]^Channel 2^Input;
                                 .q_xHV_DIS			:= 	TIIB[EL2624_01_02]^Channel 1^Output	'}
    fb_LD2_GCC : FB_MKS500; // Output tube LD2, Cold Cathode gauge

    // LD4
    {attribute 'pytmc'	  :=	' pv: LTLHN:LD4:VGC:01 '}
    {attribute 'TcLinkTo' := 	'.i_xOpnLS			:=	TIIB[EL1004_02_10]^Channel 2^Input;
                                 .i_xClsLS			:=	TIIB[EL1004_02_10]^Channel 1^Input;
                                 .q_xOPN_DO			:=	TIIB[EL2004_02_11]^Channel 1^Output'}
    fb_LD4_VGC : FB_VGC; // Gate valve, Output tube LD4 laser Table
    {attribute 'pytmc'    := 	' pv: LTLHN:LD4:PIP:01 '}
    {attribute 'TcLinkTo' := 	'.i_iPRESS			:=	TIIB[EL3064_00_11]^AI Standard Channel 1^Value;
                                 .i_xSP_DI			:= 	TIIB[EL1004_00_10]^Channel 1^Input;
                                 .q_xHVEna_DO		:= 	TIIB[EL2794_00_09]^Channel 1^Output'}
    fb_LD4_PIP : FB_PIP_Gamma; // Ion Pump, output tube LD4
    {attribute 'pytmc' 	  :=	' pv: LTLHN:LD4:GPI:01 '}
    {attribute 'TcLinkTo' := 	'.i_iPRESS_R		:=	TIIB[EL3174_03_13]^AI Standard Channel 4^Value '}
    fb_LD4_GPI : FB_MKS275; // Output tube LD4 ATM gauge
    {attribute 'pytmc' 	  :=	' pv: LTLHN:LD4:GCC:01 '}
    {attribute 'TcLinkTo' := 	'.i_iPRESS_R		:=	TIIB[EL3174_03_11]^AI Standard Channel 4^Value;
                                 .i_xHV_ON	    	:=	TIIB[EL1124_03_09]^Channel 3^Input;
                                 .i_xDisc_Active	:=	TIIB[EL1124_03_09]^Channel 4^Input;
                                 .q_xHV_DIS			:= 	TIIB[EL2624_03_02]^Channel 4^Output	'}
    fb_LD4_GCC : FB_MKS500; // Output tube LD4, Cold Cathode gauge

    // LD6
    {attribute 'pytmc'	  :=	' pv: LTLHN:LD6:VGC:01 '}
    {attribute 'TcLinkTo' := 	'.i_xOpnLS			:=	TIIB[EL1004_02_13]^Channel 4^Input;
                                 .i_xClsLS			:=	TIIB[EL1004_02_13]^Channel 3^Input;
                                 .q_xOPN_DO			:=	TIIB[EL2004_02_14]^Channel 4^Output'}
    fb_LD6_VGC : FB_VGC; // Gate valve, Output tube LD6 laser Table
    {attribute 'pytmc'    := 	' pv: LTLHN:LD6:PIP:01 '}
    {attribute 'TcLinkTo' := 	'.i_iPRESS			:=	TIIB[EL3064_00_11]^AI Standard Channel 2^Value;
                                 .i_xSP_DI			:= 	TIIB[EL1004_00_10]^Channel 2^Input;
                                 .q_xHVEna_DO		:= 	TIIB[EL2794_00_09]^Channel 2^Output'}
    fb_LD6_PIP : FB_PIP_Gamma; // Ion Pump, output tube LD6
    {attribute 'pytmc' 	  :=	' pv: LTLHN:LD6:GPI:01 '}
    {attribute 'TcLinkTo' := 	'.i_iPRESS_R		:=	TIIB[EL3174_03_13]^AI Standard Channel 3^Value '}
    fb_LD6_GPI : FB_MKS275; // Output tube LD6 ATM gauge
    {attribute 'pytmc' 	  :=	' pv: LTLHN:LD6:GCC:01 '}
    {attribute 'TcLinkTo' := 	'.i_iPRESS_R		:=	TIIB[EL3064_02_16]^AI Standard Channel 2^Value;
                                 .q_xHV_DIS	    	:=	TIIB[EL2794_02_17]^Channel 2^Input'}
    fb_LD6_GCC : FB_MKS422; // Output tube LD6, Cold Cathode gauge

    // LD8
    {attribute 'pytmc'	  :=	' pv: LTLHN:LD8:VGC:01 '}
    {attribute 'TcLinkTo' := 	'.i_xOpnLS			:=	TIIB[EL1004_02_07]^Channel 4^Input;
                                 .i_xClsLS			:=	TIIB[EL1004_02_07]^Channel 3^Input;
                                 .q_xOPN_DO			:=	TIIB[EL2004_02_08]^Channel 4^Output'}
    fb_LD8_VGC : FB_VGC; // Gate valve, Output tube LD8 laser Table
    {attribute 'pytmc'    := 	' pv: LTLHN:LD8:PIP:01 '}
    {attribute 'TcLinkTo' := 	'.i_iPRESS			:=	TIIB[EL3064_00_08]^AI Standard Channel 4^Value;
                                 .i_xSP_DI			:= 	TIIB[EL1004_00_07]^Channel 4^Input;
                                 .q_xHVEna_DO		:= 	TIIB[EL2794_00_06]^Channel 4^Output'}
    fb_LD8_PIP : FB_PIP_Gamma; // Ion Pump, output tube LD8
    {attribute 'pytmc' 	  :=	' pv: LTLHN:LD8:GPI:01 '}
    {attribute 'TcLinkTo' := 	'.i_iPRESS_R		:=	TIIB[EL3174_01_11]^AI Standard Channel 2^Value '}
    fb_LD8_GPI : FB_MKS275; // Output tube LD8 ATM gauge
    {attribute 'pytmc' 	  :=	' pv: LTLHN:LD8:GCC:01 '}
    {attribute 'TcLinkTo' := 	'.i_iPRESS_R		:=	TIIB[EL3174_01_11]^AI Standard Channel 3^Value;
                                 .i_xHV_ON	    	:=	TIIB[EL1124_01_08]^Channel 1^Input;
                                 .i_xDisc_Active	:=	TIIB[EL1124_01_08]^Channel 2^Input;
                                 .q_xHV_DIS			:= 	TIIB[EL2624_01_01]^Channel 1^Output	'}
    fb_LD8_GCC : FB_MKS500; // Output tube LD8, Cold Cathode gauge

    // LD9
    {attribute 'pytmc'	  :=	' pv: LTLHN:LD9:VGC:01 '}
    {attribute 'TcLinkTo' := 	'.i_xOpnLS			:=	TIIB[EL1004_02_06]^Channel 4^Input;
                                 .i_xClsLS			:=	TIIB[EL1004_02_06]^Channel 3^Input;
                                 .q_xOPN_DO			:=	TIIB[EL2004_02_08]^Channel 2^Output'}
    fb_LD9_VGC : FB_VGC; // Gate valve, Output tube LD9 laser Table
    {attribute 'pytmc'    := 	' pv: LTLHN:LD9:PIP:01 '}
    {attribute 'TcLinkTo' := 	'.i_iPRESS			:=	TIIB[EL3064_00_14]^AI Standard Channel 2^Value;
                                 .i_xSP_DI			:= 	TIIB[EL1004_00_13]^Channel 2^Input;
                                 .q_xHVEna_DO		:= 	TIIB[EL2794_00_12]^Channel 2^Output'}
    fb_LD9_PIP : FB_PIP_Gamma; // Ion Pump, output tube LD9
    {attribute 'pytmc' 	  :=	' pv: LTLHN:LD9:GPI:01 '}
    {attribute 'TcLinkTo' := 	'.i_iPRESS_R		:=	TIIB[EL3174_03_12]^AI Standard Channel 1^Value '}
    fb_LD9_GPI : FB_MKS275; // Output tube LD9 ATM gauge
    {attribute 'pytmc' 	  :=	' pv: LTLHN:LD9:GCC:01 '}
    {attribute 'TcLinkTo' := 	'.i_iPRESS_R		:=	TIIB[EL3174_03_10]^AI Standard Channel 1^Value;
                                 .i_xHV_ON	    	:=	TIIB[EL1124_03_06]^Channel 1^Input;
                                 .i_xDisc_Active	:=	TIIB[EL1124_03_06]^Channel 2^Input;
                                 .q_xHV_DIS			:= 	TIIB[EL2624_03_01]^Channel 1^Output	'}
    fb_LD9_GCC : FB_MKS500; // Output tube LD9, Cold Cathode gauge

    // LD10
    {attribute 'pytmc'	  :=	' pv: LTLHN:LD10:VGC:01 '}
    {attribute 'TcLinkTo' := 	'.i_xOpnLS			:=	TIIB[EL1004_02_07]^Channel 2^Input;
                                 .i_xClsLS			:=	TIIB[EL1004_02_07]^Channel 1^Input;
                                 .q_xOPN_DO			:=	TIIB[EL2004_02_08]^Channel 3^Output'}
    fb_LD10_VGC : FB_VGC; // Gate valve, Output tube LD10 laser Table
    {attribute 'pytmc'    := 	' pv: LTLHN:LD10:PIP:01 '}
    {attribute 'TcLinkTo' := 	'.i_iPRESS			:=	TIIB[EL3064_00_14]^AI Standard Channel 1^Value;
                                 .i_xSP_DI			:= 	TIIB[EL1004_00_13]^Channel 1^Input;
                                 .q_xHVEna_DO		:= 	TIIB[EL2794_00_12]^Channel 1^Output'}
    fb_LD10_PIP : FB_PIP_Gamma; // Ion Pump, output tube LD10
    {attribute 'pytmc' 	  :=	' pv: LTLHN:LD10:GPI:01 '}
    {attribute 'TcLinkTo' := 	'.i_iPRESS_R		:=	TIIB[EL3174_03_12]^AI Standard Channel 2^Value '}
    fb_LD10_GPI : FB_MKS275; // Output tube LD10 ATM gauge
    {attribute 'pytmc' 	  :=	' pv: LTLHN:LD10:GCC:01 '}
    {attribute 'TcLinkTo' := 	'.i_iPRESS_R		:=	TIIB[EL3174_03_10]^AI Standard Channel 2^Value;
                                 .i_xHV_ON	    	:=	TIIB[EL1124_03_07]^Channel 3^Input;
                                 .i_xDisc_Active	:=	TIIB[EL1124_03_07]^Channel 4^Input;
                                 .q_xHV_DIS			:= 	TIIB[EL2624_03_01]^Channel 2^Output	'}
    fb_LD10_GCC : FB_MKS500; // Output tube LD10, Cold Cathode gauge

    // LD14
    {attribute 'pytmc'	  :=	' pv: LTLHN:LD14:VGC:01 '}
    {attribute 'TcLinkTo' := 	'.i_xOpnLS			:=	TIIB[EL1004_02_10]^Channel 4^Input;
                                 .i_xClsLS			:=	TIIB[EL1004_02_10]^Channel 3^Input;
                                 .q_xOPN_DO			:=	TIIB[EL2004_02_11]^Channel 4^Output'}
    fb_LD14_VGC : FB_VGC; // Gate valve, Output tube LD14 laser Table
    {attribute 'pytmc'    := 	' pv: LTLHN:LD14:PIP:01 '}
    {attribute 'TcLinkTo' := 	'.i_iPRESS			:=	TIIB[EL3064_00_14]^AI Standard Channel 3^Value;
                                 .i_xSP_DI			:= 	TIIB[EL1004_00_13]^Channel 3^Input;
                                 .q_xHVEna_DO		:= 	TIIB[EL2794_00_12]^Channel 3^Output'}
    fb_LD14_PIP : FB_PIP_Gamma; // Ion Pump, output tube LD14
    {attribute 'pytmc' 	  :=	' pv: LTLHN:LD14:GPI:01 '}
    {attribute 'TcLinkTo' := 	'.i_iPRESS_R		:=	TIIB[EL3174_03_12]^AI Standard Channel 3^Value '}
    fb_LD14_GPI : FB_MKS275; // Output tube LD14 ATM gauge
    {attribute 'pytmc' 	  :=	' pv: LTLHN:LD14:GCC:01 '}
    {attribute 'TcLinkTo' := 	'.i_iPRESS_R		:=	TIIB[EL3174_03_10]^AI Standard Channel 3^Value;
                                 .i_xHV_ON	    	:=	TIIB[EL1124_03_07]^Channel 1^Input;
                                 .i_xDisc_Active	:=	TIIB[EL1124_03_07]^Channel 2^Input;
                                 .q_xHV_DIS			:= 	TIIB[EL2624_03_01]^Channel 3^Output	'}
    fb_LD14_GCC : FB_MKS500; // Output tube LD14, Cold Cathode gauge

    ////Bay 2 - Line Upgrade
    // LS3
    {attribute 'pytmc' 	  :=	' pv: LTLHN:LS3:GCC:01 '}
    {attribute 'TcLinkTo' := 	'.i_iPRESS_R		:=	TIIB[EL3174_01_8A]^AI Standard Channel 2^Value;
                                 .i_xHV_ON	    	:=	TIIB[EL1124_01_06]^Channel 3^Input;
                                 .i_xDisc_Active	:=	TIIB[EL1124_01_06]^Channel 4^Input;
                                 .q_xHV_DIS			:= 	TIIB[EL2624_01_01]^Channel 3^Output'}
    fb_LS3_GCC : FB_MKS500; // LS3, Cold Cathode gauge
    {attribute 'pytmc' 	  :=	' pv: LTLHN:LS3:GPI:01 '}
    {attribute 'TcLinkTo' := 	'.i_iPRESS_R		:=	TIIB[EL3174_01_11]^AI Standard Channel 4^Value '}
    fb_LS3_GPI : FB_MKS275; // LS3 Pirani gauge
    {attribute 'pytmc'	  :=	' pv: LTLHN:LS3:VGC:01 '}
    {attribute 'TcLinkTo' := 	'.i_xOpnLS			:=	TIIB[EL1004_00_16]^Channel 1^Input;
                                 .i_xClsLS			:=	TIIB[EL1004_00_16]^Channel 2^Input;
                                 .q_xOPN_DO			:=	TIIB[EL2004_00_17]^Channel 1^Output'}
    fb_LS3_VGC : FB_VGC; // Gate valve
    {attribute 'pytmc'    := 	' pv: LTLHN:LS3:PIP:01 '}
    {attribute 'TcLinkTo' := 	'.i_iPRESS			:=	TIIB[EL3064_01_15]^AI Standard Channel 1^Value;
                                 .i_xSP_DI			:= 	TIIB[EL1004_01_16]^Channel 1^Input;
                                 .q_xHVEna_DO		:= 	TIIB[EL2794_01_17]^Channel 1^Output'}
    fb_LS3_PIP : FB_PIP_Gamma; // Ion Pump
    //LS4
    {attribute 'pytmc' 	  :=	' pv: LTLHN:LS4:GCC:01 '}
    {attribute 'TcLinkTo' := 	'.i_iPRESS_R		:=	TIIB[EL3174_01_8A]^AI Standard Channel 3^Value;
                                 .i_xHV_ON	    	:=	TIIB[EL1124_01_08]^Channel 3^Input;
                                 .i_xDisc_Active	:=	TIIB[EL1124_01_08]^Channel 4^Input;
                                 .q_xHV_DIS			:= 	TIIB[EL2624_01_01]^Channel 4^Output	'}
    fb_LS4_GCC : FB_MKS500; // LS4, Cold Cathode gauge
    {attribute 'pytmc' 	  :=	' pv: LTLHN:LS4:GPI:01 '}
    {attribute 'TcLinkTo' := 	'.i_iPRESS_R		:=	TIIB[EL3174_01_09]^AI Standard Channel 3^Value '}
    fb_LS4_GPI : FB_MKS275; // LS4 Pirani gauge
    {attribute 'pytmc'	  :=	' pv: LTLHN:LS4:VGC:01 '}
    {attribute 'TcLinkTo' := 	'.i_xOpnLS			:=	TIIB[EL1004_00_16]^Channel 3^Input;
                                 .i_xClsLS			:=	TIIB[EL1004_00_16]^Channel 4^Input;
                                 .q_xOPN_DO			:=	TIIB[EL2004_00_17]^Channel 2^Output'}
    fb_LS4_VGC : FB_VGC; // Gate valve
    {attribute 'pytmc'    := 	' pv: LTLHN:LS4:PIP:01 '}
    {attribute 'TcLinkTo' := 	'.i_iPRESS			:=	TIIB[EL3064_01_15]^AI Standard Channel 2^Value;
                                 .i_xSP_DI			:= 	TIIB[EL1004_01_16]^Channel 2^Input;
                                 .q_xHVEna_DO		:= 	TIIB[EL2794_01_17]^Channel 2^Output'}
    fb_LS4_PIP : FB_PIP_Gamma; // Ion Pump
    //LS6
    {attribute 'pytmc' 	  :=	' pv: LTLHN:LS6:GCC:01 '}
    {attribute 'TcLinkTo' := 	'.i_iPRESS_R		:=	TIIB[EL3064_02_16]^AI Standard Channel 1^Value;
                                 .q_xHV_DIS	    	:=	TIIB[EL2794_02_17]^Channel 1^Input'}
    fb_LS6_GCC : FB_MKS422; // LS6, Cold Cathode gauge

    {attribute 'pytmc' 	  :=	' pv: LTLHN:LS6:GPI:01 '}
    {attribute 'TcLinkTo' := 	'.i_iPRESS_R		:=	TIIB[EL3174_01_09]^AI Standard Channel 3^Value '}
    fb_LS6_GPI : FB_MKS275; // LS6 Pirani gauge
    {attribute 'pytmc'	  :=	' pv: LTLHN:LS6:VGC:01 '}
    {attribute 'TcLinkTo' := 	'.i_xOpnLS			:=	TIIB[EL1004_02_13]^Channel 1^Input;
                                 .i_xClsLS			:=	TIIB[EL1004_02_13]^Channel 2^Input;
                                 .q_xOPN_DO			:=	TIIB[EL2004_02_14]^Channel 1^Output'}
    fb_LS6_VGC : FB_VGC; // Gate valve
    {attribute 'pytmc'    := 	' pv: LTLHN:LS6:PIP:01 '}
    {attribute 'TcLinkTo' := 	'.i_iPRESS			:=	TIIB[EL3064_01_15]^AI Standard Channel 3^Value;
                                 .i_xSP_DI			:= 	TIIB[EL1004_01_16]^Channel 3^Input;
                                 .q_xHVEna_DO		:= 	TIIB[EL2794_01_17]^Channel 3^Output'}
    fb_LS6_PIP : FB_PIP_Gamma; // Ion Pump
    //Preemptive Arbiter Content
    g_fbArbiter    :   FB_Arbiter(1);

END_VAR

// ---- POUs/PRG_VALVES.TcPOU
PROGRAM PRG_VALVES
VAR

END_VAR

(* Switchbox valves *)
fb_PP_VGC(
    i_stUSG := fb_PP_GCC.IG,
    i_stDSG := fb_DP_GCC.IG,
    i_xDis_DPIlk := FALSE,
    i_xEPS_OK := TRUE,
    i_xPMPS_OK := TRUE,
    i_xExt_OK := TRUE,
    i_xOverrideMode := xSystemOverrideMode_BTS,
    io_fbFFHWO := g_FFOut,
    fbArbiter := g_fbArbiter
);

fb_PP_VVC(
    i_xExtILK_OK := fb_PP_VGC.M_IsClosed(),
    i_xOverrideMode := xSystemOverrideMode_BTS
);

GVL_BTS_VAC.fb_PP_VRC_1(
    i_xExtILK_OK := TRUE,
    i_xOverrideMode := xSystemOverrideMode_BTS
);

GVL_BTS_VAC.fb_PP_VRC_2(
    i_xExtILK_OK := TRUE,
    i_xOverrideMode := xSystemOverrideMode_BTS
);

fb_VP_VVC_1(
    i_xExtILK_OK := TRUE,
    i_xOverrideMode := xSystemOverrideMode_BTS
);

fb_VP_VVC_2(
    i_xExtILK_OK := TRUE
);

// Vent manifold valve - interlock logic with slow or fast vent
IF (fb_PP_PMF.q_stPump.eState <> E_PumpState.pumpSTOPPED)  THEN  // Condition to evaluate if Roughing Pump is ON
    fb_VP_VVC_4.i_xExtILK_OK := FALSE;
    fb_VP_VVC_2.i_xExtILK_OK := FALSE;
    fb_VP_VVC_1.i_xExtILK_OK := FALSE;
ELSE
    fb_VP_VVC_4.i_xExtILK_OK := TRUE;
    fb_VP_VVC_2.i_xExtILK_OK := TRUE;
    fb_VP_VVC_1.i_xExtILK_OK := TRUE;
        IF (fb_VP_VVC_2.iq_stValve.q_xOPN_DO OR fb_VP_VVC_1.iq_stValve.q_xOPN_DO) THEN
            fb_VP_VVC_4.M_Set_OPN_SW(TRUE);
        ELSE
            fb_VP_VVC_4.M_Set_OPN_SW(FALSE);
        END_IF
END_IF

fb_VP_VVC_4(
    i_xOverrideMode := xSystemOverrideMode_BTS
);

// Turbo Isolation valve - Interlocked with turbo pump operation

//Roughing Pump function block
fb_PP_VRC_4(
    i_xExtILK_OK := (fb_PP_PMF.q_stPump.eState = E_PumpState.pumpRUNNING) OR (fb_PP_PMF.q_stPump.eState = E_PumpState.pumpSTARTING),
    i_xOverrideMode := xSystemOverrideMode_BTS
);

/////Forcing Valve to OPEN when PUMP is RUNNING
//Required by Laser Hall
IF (fb_PP_PMF.q_stPump.eState = E_PumpState.pumpRUNNING or fb_PP_PMF.q_stPump.eState = E_PumpState.pumpSTARTING)THEN
    fb_PP_VRC_4.M_Set_OPN_SW(TRUE);
END_IF

(* Transport Tube vavles *)
// LS1
fb_LS1_VGC(
    i_stUSG := fb_LS1_GCC.IG,
    i_stDSG := fb_DP_GCC.IG,
    i_xDis_DPIlk := FALSE,
    i_xEPS_OK := TRUE,
    i_xPMPS_OK := TRUE,
    i_xExt_OK := TRUE,
    i_xOverrideMode := xSystemOverrideMode_BTS,
    io_fbFFHWO := g_FFOut,
    fbArbiter := g_fbArbiter,
);

// LS5
fb_LS5_VGC(
    i_stUSG := fb_LS5_GPI.PG,
    i_stDSG := fb_DP_GPI.PG,
    i_xDis_DPIlk := FALSE,
    i_xEPS_OK := TRUE,
    i_xPMPS_OK := TRUE,
    i_xExt_OK := TRUE,
    i_xOverrideMode := xSystemOverrideMode_BTS,
    io_fbFFHWO := g_FFOut,
    fbArbiter := g_fbArbiter
);

// LS8
fb_LS8_VGC(
    i_stUSG := fb_LS8_GCC.IG,
    i_stDSG := fb_DP_GCC.IG,
    i_xDis_DPIlk := FALSE,
    i_xEPS_OK := TRUE,
    i_xPMPS_OK := TRUE,
    i_xExt_OK := TRUE,
    i_xOverrideMode := xSystemOverrideMode_BTS,
    io_fbFFHWO := g_FFOut,
    fbArbiter := g_fbArbiter
);

// LD2
fb_LD2_VGC(
    i_stUSG := fb_LD2_GCC.IG,
    i_stDSG := fb_DP_GCC.IG,
    i_xDis_DPIlk := FALSE,
    i_xEPS_OK := TRUE,
    i_xPMPS_OK := TRUE,
    i_xExt_OK := TRUE,
    i_xOverrideMode := xSystemOverrideMode_BTS,
    io_fbFFHWO := g_FFOut,
    fbArbiter := g_fbArbiter
);

// LD4
fb_LD4_VGC(
    i_stUSG := fb_LD4_GCC.IG,
    i_stDSG := fb_DP_GCC.IG,
    i_xDis_DPIlk := FALSE,
    i_xEPS_OK := TRUE,
    i_xPMPS_OK := TRUE,
    i_xExt_OK := TRUE,
    i_xOverrideMode := xSystemOverrideMode_BTS,
    io_fbFFHWO := g_FFOut,
    fbArbiter := g_fbArbiter
);

// LD6
fb_LD6_VGC(
    i_stUSG := fb_LD6_GCC.IG,
    i_stDSG := fb_DP_GCC.IG,
    i_xDis_DPIlk := FALSE,
    i_xEPS_OK := TRUE,
    i_xPMPS_OK := TRUE,
    i_xExt_OK := TRUE,
    i_xOverrideMode := xSystemOverrideMode_BTS,
    io_fbFFHWO := g_FFOut,
    fbArbiter := g_fbArbiter
);

// LD8
fb_LD8_VGC(
    i_stUSG := fb_LD8_GCC.IG,
    i_stDSG := fb_DP_GCC.IG,
    i_xDis_DPIlk := FALSE,
    i_xEPS_OK := TRUE,
    i_xPMPS_OK := TRUE,
    i_xExt_OK := TRUE,
    i_xOverrideMode := xSystemOverrideMode_BTS,
    io_fbFFHWO := g_FFOut,
    fbArbiter := g_fbArbiter
);

// LD9
fb_LD9_VGC(
    i_stUSG := fb_LD9_GCC.IG,
    i_stDSG := fb_DP_GCC.IG,
    i_xDis_DPIlk := FALSE,
    i_xEPS_OK := TRUE,
    i_xPMPS_OK := TRUE,
    i_xExt_OK := TRUE,
    i_xOverrideMode := xSystemOverrideMode_BTS,
    io_fbFFHWO := g_FFOut,
    fbArbiter := g_fbArbiter
);

// LD10
fb_LD10_VGC(
    i_stUSG := fb_LD10_GCC.IG,
    i_stDSG := fb_DP_GCC.IG,
    i_xDis_DPIlk := FALSE,
    i_xEPS_OK := TRUE,
    i_xPMPS_OK := TRUE,
    i_xExt_OK := TRUE,
    i_xOverrideMode := xSystemOverrideMode_BTS,
    io_fbFFHWO := g_FFOut,
    fbArbiter := g_fbArbiter
);

// LD14
fb_LD14_VGC(
    i_stUSG := fb_LD14_GCC.IG,
    i_stDSG := fb_DP_GCC.IG,
    i_xDis_DPIlk := FALSE,
    i_xEPS_OK := TRUE,
    i_xPMPS_OK := TRUE,
    i_xExt_OK := TRUE,
    i_xOverrideMode := xSystemOverrideMode_BTS,
    io_fbFFHWO := g_FFOut,
    fbArbiter := g_fbArbiter
);


//// LS3
fb_LS3_VGC(
    i_stUSG := fb_LS3_GPI.PG,
    i_stDSG := fb_DP_GPI.PG,
    i_xDis_DPIlk := FALSE,
    i_xEPS_OK := TRUE,
    i_xPMPS_OK := TRUE,
    i_xExt_OK := TRUE,
    i_xOverrideMode := xSystemOverrideMode_BTS,
    io_fbFFHWO := g_FFOut,
    fbArbiter := g_fbArbiter
);

// LS4
fb_LS4_VGC(
    i_stUSG := fb_LS4_GPI.PG,
    i_stDSG := fb_DP_GPI.PG,
    i_xDis_DPIlk := FALSE,
    i_xEPS_OK := TRUE,
    i_xPMPS_OK := TRUE,
    i_xExt_OK := TRUE,
    i_xOverrideMode := xSystemOverrideMode_BTS,
    io_fbFFHWO := g_FFOut,
    fbArbiter := g_fbArbiter
);

// LS6
fb_LS6_VGC(
    i_stUSG := fb_LS6_GPI.PG,
    i_stDSG := fb_DP_GPI.PG,
    i_xDis_DPIlk := FALSE,
    i_xEPS_OK := TRUE,
    i_xPMPS_OK := TRUE,
    i_xExt_OK := TRUE,
    i_xOverrideMode := xSystemOverrideMode_BTS,
    io_fbFFHWO := g_FFOut,
    fbArbiter := g_fbArbiter
);

END_PROGRAM
